// TIA Portal V19 export
TYPE "udt_FlyingCarriage_Config"
   STRUCT
      SLS_VEL { ExternalVisible := 'False'; ExternalWritable := 'False'; S7_SetPoint := 'True'} : LReal := 3.0;
      DelayMissingCondition { ExternalVisible := 'False'; ExternalWritable := 'False'; S7_SetPoint := 'True'} : Time := T#3S;
      Fan { ExternalVisible := 'False'; ExternalWritable := 'False'} : Struct
         Exist { S7_SetPoint := 'True'} : Bool := TRUE;
         DelayOff { S7_SetPoint := 'True'} : Time := T#15M;
      END_STRUCT;
   END_STRUCT;
END_TYPE
